// Mitsubishi GX Works2 project: HELLOWORLD2709.gx3   PLC: Q03UDV

PROGRAM MAIN
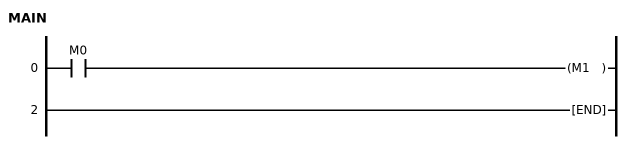
0     LD      M0
      OUT     M1
2     END
END_PROGRAM
